FUNCTION_BLOCK fbreturn5
VAR_INPUT
END_VAR
VAR_OUTPUT
END_VAR
VAR
END_VAR

END_FUNCTION_BLOCK

(* stored: Version 1.1.0.1, ProductVersion 3.1.4024.12
   POU fbreturn5: Id {9c594cfb-17d1-49ed-93c8-d821f6533f37}, SpecialFunc None *)
